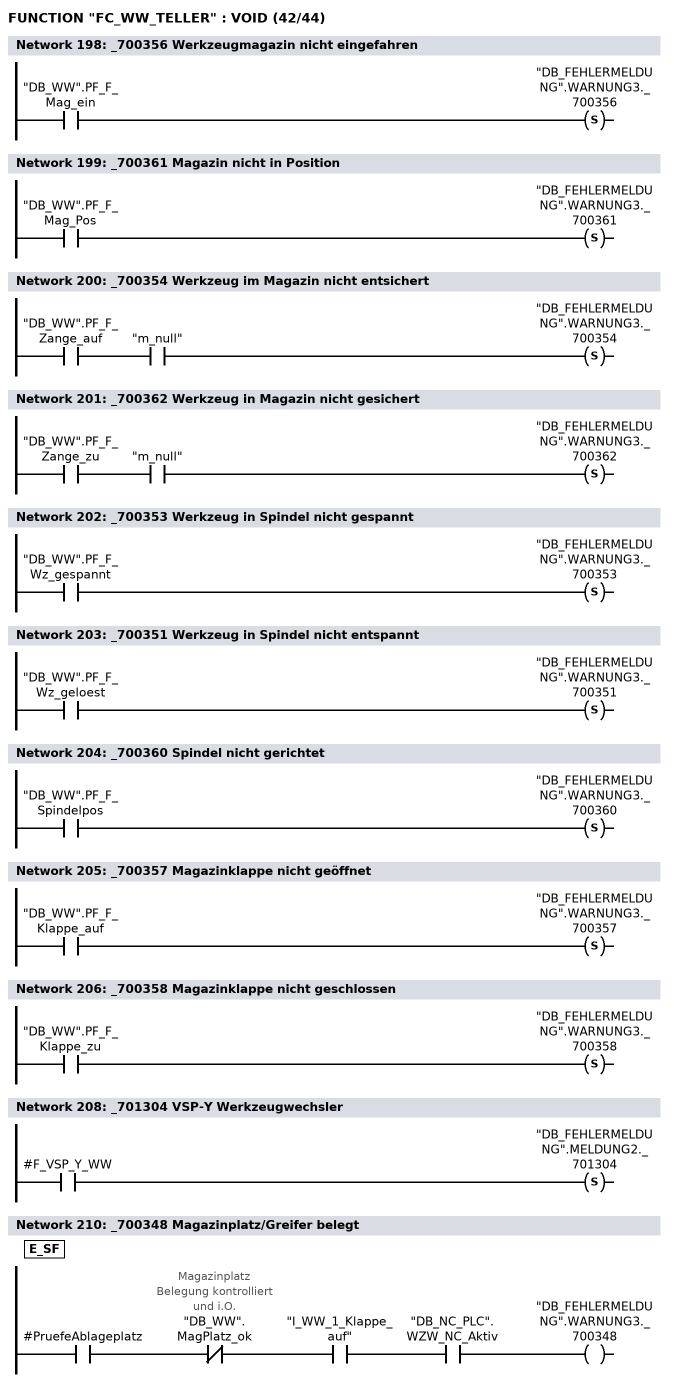

      U     "DB_WW".PF_F_Mag_ein;
      S     "DB_FEHLERMELDUNG".WARNUNG3._700356;

NETWORK
TITLE =_700361 Magazin nicht in Position

      U     "DB_WW".PF_F_Mag_Pos;
      S     "DB_FEHLERMELDUNG".WARNUNG3._700361;

NETWORK
TITLE =_700354 Werkzeug im Magazin nicht entsichert

      U     "DB_WW".PF_F_Zange_auf;
      U     "m_null";
      S     "DB_FEHLERMELDUNG".WARNUNG3._700354;

NETWORK
TITLE =_700362 Werkzeug in Magazin nicht gesichert

      U     "DB_WW".PF_F_Zange_zu;
      U     "m_null";
      S     "DB_FEHLERMELDUNG".WARNUNG3._700362;

NETWORK
TITLE =_700353 Werkzeug in Spindel nicht gespannt

      U     "DB_WW".PF_F_Wz_gespannt;
      S     "DB_FEHLERMELDUNG".WARNUNG3._700353;

NETWORK
TITLE =_700351 Werkzeug in Spindel nicht entspannt

      U     "DB_WW".PF_F_Wz_geloest;
      S     "DB_FEHLERMELDUNG".WARNUNG3._700351;

NETWORK
TITLE =_700360 Spindel nicht gerichtet

      U     "DB_WW".PF_F_Spindelpos;
      S     "DB_FEHLERMELDUNG".WARNUNG3._700360;

NETWORK
TITLE =_700357 Magazinklappe nicht geöffnet

      U     "DB_WW".PF_F_Klappe_auf;
      S     "DB_FEHLERMELDUNG".WARNUNG3._700357;
NETWORK
TITLE =_700358 Magazinklappe nicht geschlossen

      U     "DB_WW".PF_F_Klappe_zu;
      S     "DB_FEHLERMELDUNG".WARNUNG3._700358;

NETWORK
TITLE =_701302 Spindel leer
//  U     "DB_WW".PF_F_Spindel_leer
//  S     "DB_FEHLERMELDUNG".MELDUNG2._701302    // Spindel leer


NETWORK
TITLE =_701304 VSP-Y Werkzeugwechsler

      U     #F_VSP_Y_WW;
      S     "DB_FEHLERMELDUNG".MELDUNG2._701304;
NETWORK
TITLE ========= Sonstige Fehler- Betriebsmeldungen ===========



NETWORK
TITLE =_700348 Magazinplatz/Greifer belegt

E_SF: U     #PruefeAblageplatz;
      UN    "DB_WW".MagPlatz_ok; // Magazinplatz Belegung kontrolliert und i.O.
      U     "I_WW_1_Klappe_auf";
      U     "DB_NC_PLC".WZW_NC_Aktiv;

      =     "DB_FEHLERMELDUNG".WARNUNG3._700348;
NETWORK
TITLE =_700349 Magazinplatz/Greifer leer
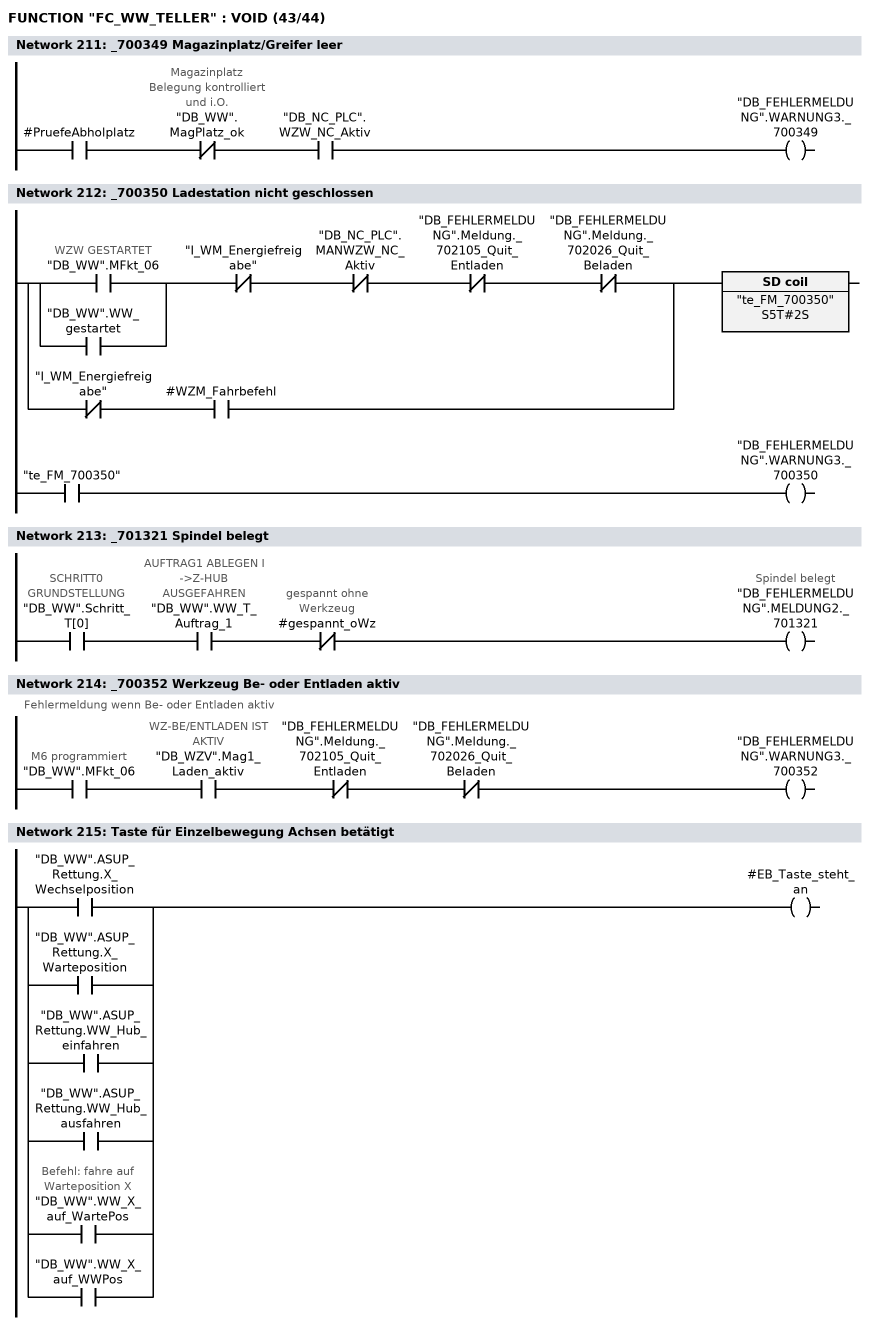

      U     #PruefeAbholplatz;
      UN    "DB_WW".MagPlatz_ok; // Magazinplatz Belegung kontrolliert und i.O.
      U     "DB_NC_PLC".WZW_NC_Aktiv;
      =     "DB_FEHLERMELDUNG".WARNUNG3._700349;

NETWORK
TITLE =_700350 Ladestation nicht geschlossen

      U(    ;
      U(    ; // M6
      O     "DB_WW".MFkt_06; // WZW GESTARTET
      O     "DB_WW".WW_gestartet;
      )     ; // Wz-Magazintür geschlossen
      UN    "I_WM_Energiefreigabe";
      UN    "DB_NC_PLC".MANWZW_NC_Aktiv;
      UN    "DB_FEHLERMELDUNG".Meldung._702105_Quit_Entladen;
      UN    "DB_FEHLERMELDUNG".Meldung._702026_Quit_Beladen;
      O     ; // Wz-Magazintür geschlossen
      UN    "I_WM_Energiefreigabe";
      U     #WZM_Fahrbefehl;

      )     ;
      L     S5T#2S;
      SE    "te_FM_700350";
      NOP   0;
      NOP   0;
      NOP   0;
      U     "te_FM_700350";
      =     "DB_FEHLERMELDUNG".WARNUNG3._700350;
NETWORK
TITLE =_701321 Spindel belegt

      U     "DB_WW".Schritt_T[0]; // SCHRITT0 GRUNDSTELLUNG
      U     "DB_WW".WW_T_Auftrag_1; // AUFTRAG1 ABLEGEN I ->Z-HUB AUSGEFAHREN
      UN    #gespannt_oWz; // gespannt ohne Werkzeug
      =     "DB_FEHLERMELDUNG".MELDUNG2._701321; // Spindel belegt

NETWORK
TITLE =_700352 Werkzeug Be- oder Entladen aktiv
// Fehlermeldung wenn Be- oder Entladen aktiv
      U     "DB_WW".MFkt_06; // M6 programmiert
      U     "DB_WZV".Mag1_Laden_aktiv; // WZ-BE/ENTLADEN IST AKTIV
      UN    "DB_FEHLERMELDUNG".Meldung._702105_Quit_Entladen;
      UN    "DB_FEHLERMELDUNG".Meldung._702026_Quit_Beladen;
      =     "DB_FEHLERMELDUNG".WARNUNG3._700352;

NETWORK
TITLE =Taste für Einzelbewegung Achsen betätigt

      O     "DB_WW".ASUP_Rettung.X_Wechselposition;
      O     "DB_WW".ASUP_Rettung.X_Warteposition;
      O     "DB_WW".ASUP_Rettung.WW_Hub_einfahren;
      O     "DB_WW".ASUP_Rettung.WW_Hub_ausfahren;
      O     "DB_WW".WW_X_auf_WartePos; // Befehl: fahre auf Warteposition X
      O     "DB_WW".WW_X_auf_WWPos;
      =     #EB_Taste_steht_an;

NETWORK
TITLE =_700550 EINLESESPERRE, Werkzeugwechsel
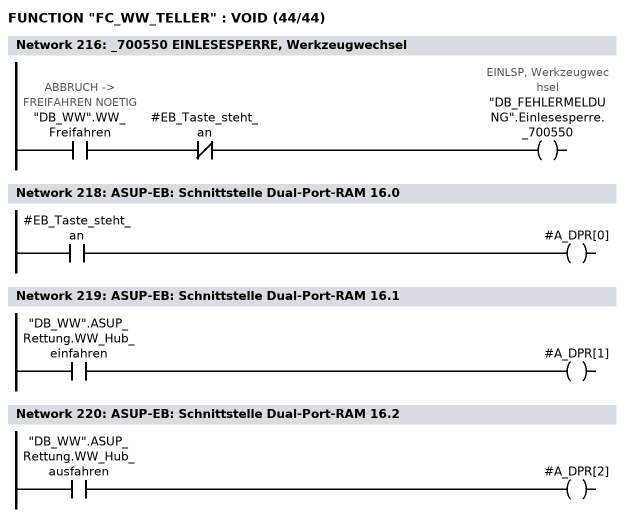

      U     "DB_WW".WW_Freifahren; // ABBRUCH -> FREIFAHREN NOETIG
      UN    #EB_Taste_steht_an;
      =     "DB_FEHLERMELDUNG".Einlesesperre._700550; // EINLSP, Werkzeugwechsel

NETWORK
TITLE ========= ASUP Einzelbewegung Achsen ========



NETWORK
TITLE =ASUP-EB: Schnittstelle Dual-Port-RAM 16.0

      U     #EB_Taste_steht_an;
      =     #A_DPR[0];

NETWORK
TITLE =ASUP-EB: Schnittstelle Dual-Port-RAM 16.1

      U     "DB_WW".ASUP_Rettung.WW_Hub_einfahren;
      =     #A_DPR[1];

NETWORK
TITLE =ASUP-EB: Schnittstelle Dual-Port-RAM 16.2

      U     "DB_WW".ASUP_Rettung.WW_Hub_ausfahren;
      =     #A_DPR[2];

NETWORK
TITLE =ASUP-EB: Schnittstelle Dual-Port-RAM 16.3

      O     "DB_WW".WW_X_auf_WartePos; // Befehl: fahre auf Warteposition X
      O     "DB_WW".ASUP_Rettung.X_Warteposition;
      FP    "HM_PI_X_AX_auf_WFKpos";
      SPBN  n20e;

      SET   ;
      S     "Start_ASUP_Machine_Nr.1";
      L     2;
      T     "DB_NC_PLC".Rettung_FktNr;

n20e: NOP   0;


//  =     #A_DPR[3]

NETWORK
TITLE =ASUP-EB: Schnittstelle Dual-Port-RAM 16.4

      O     "DB_WW".WW_X_auf_WWPos;
      O     "DB_WW".ASUP_Rettung.X_Wechselposition;
      FP    "HM_PI_Bew_68_Minus";
      SPBN  n22e;

      SET   ;
      S     "Start_ASUP_Machine_Nr.1";
      L     1;
      T     "DB_NC_PLC".Rettung_FktNr;

n22e: U     "DB_EINRICHTFUNKTION".Bewegung_15_Minus; //Vert-Achse auf Wechselposition
      FP    "HM_PI_Bew_69_Plus";
      SPBN  n20c;
      S     "Start_ASUP_Machine_Nr.1";
      L     3;
      T     "DB_NC_PLC".Rettung_FktNr;

n20c: U     "DB_EINRICHTFUNKTION".Bewegung_16_Plus; //Spindel auf Wechselposition
      U     "M_Leistung_Steht_an";
      U     "I_WZ_SPA_gespannt";
      FP    "HM_PI_Bew_70_Plus";
      SPBN  n20z;
      S     "Start_ASUP_Machine_Nr.1";
      L     4;
      T     "DB_NC_PLC".Rettung_FktNr;


n20z: NOP   0;




NETWORK
TITLE =Asup abbrechen wenn Taste wieder losgelassen wird
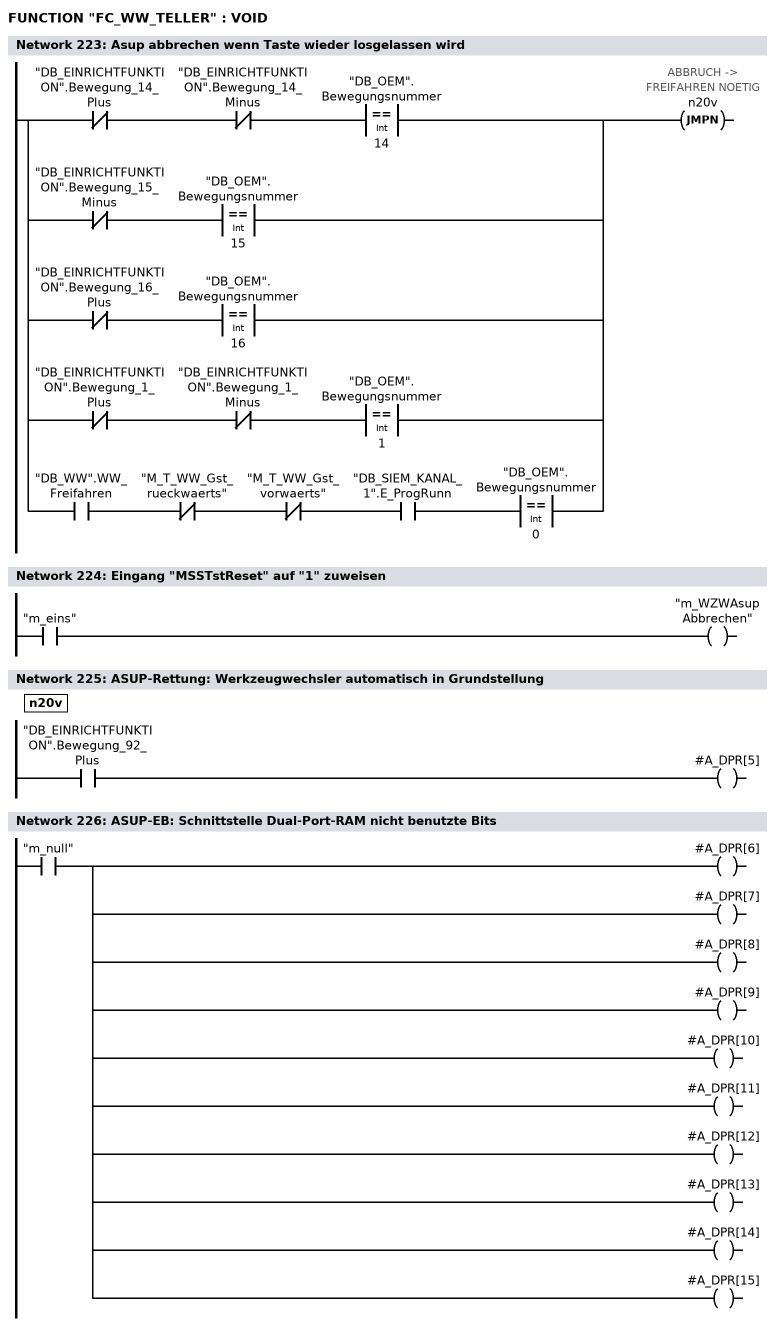

      UN    "DB_EINRICHTFUNKTION".Bewegung_14_Plus;
      UN    "DB_EINRICHTFUNKTION".Bewegung_14_Minus;
      U(    ;
      L     "DB_OEM".Bewegungsnummer;
      L     14;
      ==I   ;
      )     ;
      O     ;
      UN    "DB_EINRICHTFUNKTION".Bewegung_15_Minus;
      U(    ;
      L     "DB_OEM".Bewegungsnummer;
      L     15;
      ==I   ;
      )     ;
      O     ;
      UN    "DB_EINRICHTFUNKTION".Bewegung_16_Plus;
      U(    ;
      L     "DB_OEM".Bewegungsnummer;
      L     16;
      ==I   ;
      )     ;
      O     ;
      UN    "DB_EINRICHTFUNKTION".Bewegung_1_Plus;
      UN    "DB_EINRICHTFUNKTION".Bewegung_1_Minus;
      U(    ;
      L     "DB_OEM".Bewegungsnummer;
      L     1;
      ==I   ;
      )     ;
      O     ;
      U     "DB_WW".WW_Freifahren;
      UN    "M_T_WW_Gst_rueckwaerts";
      UN    "M_T_WW_Gst_vorwaerts";
      U     "DB_SIEM_KANAL_1".E_ProgRunn;
      U(    ;
      L     "DB_OEM".Bewegungsnummer;
      L     0;
      ==I   ;
      )     ;
      SPBN  n20v; // ABBRUCH -> FREIFAHREN NOETIG
NETWORK
TITLE =Eingang "MSSTstReset" auf "1" zuweisen

      U     "m_eins";
      =     "m_WZWAsupAbbrechen";
NETWORK
TITLE =ASUP-Rettung: Werkzeugwechsler automatisch in Grundstellung

n20v: U     "DB_EINRICHTFUNKTION".Bewegung_92_Plus;
      =     #A_DPR[5];

NETWORK
TITLE =ASUP-EB: Schnittstelle Dual-Port-RAM nicht benutzte Bits

      U     "m_null";
      =     #A_DPR[6];
      =     #A_DPR[7];
      =     #A_DPR[8];
      =     #A_DPR[9];
      =     #A_DPR[10];
      =     #A_DPR[11];
      =     #A_DPR[12];
      =     #A_DPR[13];
      =     #A_DPR[14];
      =     #A_DPR[15];

NETWORK
TITLE =ASUP-EB: Aufruf Kanal-DB für FC21

      AUF   "DB_SIEM_KANAL_1";

NETWORK
TITLE =ASUP-EB: Übergabe an DUAL-PORT-RAM

      U     "m_eins";
      =     L     24.0;
      BLD   103;
      CALL "FC_SIEM_PLC_NCK" (
           Enable                   := L     24.0,
           Funct                    := B#16#4,
           S7Var                    := #A_DPR,
           IVAR1                    := 16,
           IVAR2                    := -1,
           Error                    := #FC21_Error,
           ErrCode                  := #FC21_ErrCode);
      NOP   0;
NETWORK
TITLE =ASUP-EB: Start für Einzelbewegung Achsen

      U     #EB_Taste_steht_an;
      FP    "DB_WW".ASUP_Rettung.PF_Start;
      =     "DB_SIEM_NCK".A_Set_Inp8;

NETWORK
TITLE =GRundstelltung Radmagazin



NETWORK
TITLE ============= Signale an andere Module =============
//  dieses Netzwerk ins Saftey Modul, da CS kein Profisafe
//
//      U     "DB_WW".WW_Gst; // WZW IN GRUNDSTELLUNG
//      U     "I_WW_1_Klappe_zu"; // Magazinklappe geschlossen
//      UN    "DB_WW".MFkt_06;
//      UN    "DB_WW".WW_gestartet;
//      =     "DB_HR".SI.WW_nicht_aktiv;


NETWORK
TITLE =Übergabe der Schrittnummer Werkzeugwechsel an HMI

      CALL "FC_UT_BIT_TO_DEZ" (
           Bit_Zeiger               := "DB_WW".Schritt_T,
           Anzahl_Byte              := 2,
           Dezimal                  := "DB_OEM".WZW_Ablauf_Schritt);


NETWORK
TITLE =An NC: PLC-Freigabe Werkzeugwechsel

      U     "I_WW_Freigabe"; // WZW Freigabe 1-Signal
      U     "M_WZW_Grdst"; // und der WZW ist in Grundstellung
      U     "I_AL_Kabine_Verriegelt";
      UN    "M_3Te_Betriebsart";
      UN    "M_4Te_Betriebsart";
      UN    "M_Einrichtbetrieb";
      U     "M_Leistung_Steht_an";
      UN    "MX_TDS_Aktiv";
      U(    ;
      U     "I_LA_eingeschwenkt";
      O(    ;
      L     "DB_PLC_MD_DB20".UDInt._032_ANWAHL_WZVERMESSUNG;
      L     0;
      ==I   ;
      )     ;
      O(    ;
      TAK   ;
      L     3;
      ==I   ;
      )     ;
      )     ;
      UN    "DB_OUT".AmxLockToolChanger;
      =     "DB_NC_PLC".WZW_PLC_Freigabe; // Alle Bedingungen ok Startsignal an NC
NETWORK
TITLE =An NC: Rad in Wechselstellung nach Be./Enladen an Beladestelle
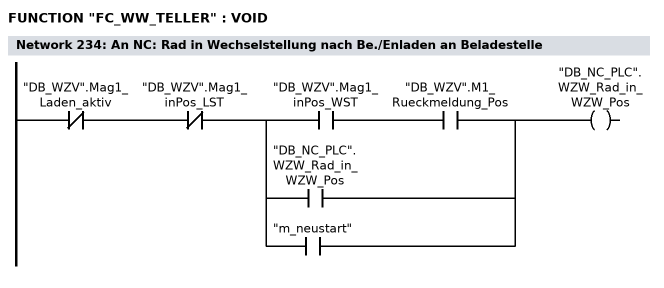

      UN    "DB_WZV".Mag1_Laden_aktiv;
      UN    "DB_WZV".Mag1_inPos_LST;
      U(    ;


      U     "DB_WZV".Mag1_inPos_WST;
      U     "DB_WZV".M1_Rueckmeldung_Pos;
      O     "DB_NC_PLC".WZW_Rad_in_WZW_Pos;
      O     "m_neustart";
      )     ;
      =     "DB_NC_PLC".WZW_Rad_in_WZW_Pos;
END_FUNCTION

